FUNCTION_BLOCK Q_GraphicsContext (* Command Graphics Context ( Part 6 - F.56 ) *)
  (* Standard: ISO 11783-6; Description: Copyright (c) 2022 HR Agrartechnik GmbH This program and the accompanying materials are made available under the terms of the Eclipse Public License 2.0 which is available at https://www.eclipse.org/legal/epl-2.0/ SPDX-License-Identifier: EPL-2.0 see Description Tab *)
  (* Version 1.0, 2022-07-08, Franz Höpfinger, HR Agrartechnik GmbH *)
  PACKAGE isobus::UT::Q;
  IMPORT isobus::UT::Q::const::IDs::ID_NULL;
  (* Documentation:
  Command Graphics Context ( Part 6 - F.56 )
   This command is used to manipulate a graphics Context object (only on version 4 or later VTs).
   Valid Object IDs
   A graphics context Object ID is valid if it falls within the following ISO 11783-6 ID range:
    - GraphicsContextObject: 36000 – 36999
    ID_NULL (65535) is not a command target but can be used in INIT to deactivate the FB. Any ID outside this range is invalid for commanding.
   Activate / Deactivate
   The FB is deactivated by default. It becomes active when INIT provides a valid graphics context Object ID. Sending INIT with ID_NULL (65535) deactivates the FB again. This toggle can be repeated arbitrarily.
    - INIT + ID_NULL (65535): FB deactivated, STATUS="DEACTIVATED", s16result=VT_E_DEACTIVATED (-40)
   - INIT + valid graphics context ID: FB activated, STATUS="initialized", s16result=VT_E_NO_ERR (0). If a REQ was buffered before, it is executed immediately.
   - INIT + invalid ID: STATUS="ERROR: Invalid Object ID (not a graphics context object)", s16result=VT_E_INVALID_OBJECT_ID (-132)
    REQ Handling
    - REQ before any INIT: Buffered, STATUS="Buffered: INIT not yet completed", s16result=VT_E_NOT_READY (-131)
   - REQ while deactivated (INIT came with NULL or invalid ID): STATUS shows the actual deactivation reason, s16result=VT_E_DEACTIVATED (-40) or VT_E_INVALID_OBJECT_ID (-132)
   - REQ while active: Command sent to VT, result reflected in CNF
    param[in] {objectID, uint16_t}
   Object ID of a Graphics Context object. Use ID_NULL (65535) to deactivate the FB. Use a valid graphics context object ID to activate.
   param[in] {SubCommandID, uint8_t}
   Sub-Command ID
   param[in] {ParameterSubCommandID_Byte, const uint8_t *}
   Parameters based on sub-command ID byte
   param[in] {LenBytes, uint16_t}
   Length in bytes of parameter list
   Return Values (s16result):
   int16_t
    - VT_E_NO_ERR (0) - OK
   - VT_E_DEACTIVATED (-40) - FB deactivated (INIT received with ID_NULL)
   - VT_E_INVALID_OBJECT_ID (-132) - Object ID is invalid (not a graphics context object)
   - VT_E_NOT_READY (-131) - Buffered: INIT not yet completed
   - VT_E_OVERFLOW (-6) - buffer overflow
   - VT_E_NOACT (-8) - Command not possible in current state
   - VT_E_NO_INSTANCE (-21) - No VT client available
   - VT_E_ISO_INSTANCE_INVALID (-129) - Identifier for instance (connection) invalid
   - VT_E_NOT_ALIVE (-130) - Identifier for instance valid, but VT Dead.
    Note
    - Function uses string buffer ( Parameterlist has to be smaller than ISO_VTC_CMD_STR_MAX_LENGTH )
  *)
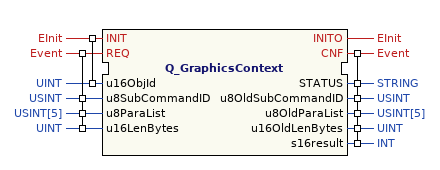
  EVENT_INPUT
    INIT : EInit WITH u16ObjId; (* Service Initialization *)
    REQ WITH u8SubCommandID, u8ParaList, u16LenBytes; (* Service Request *)
  END_EVENT
  EVENT_OUTPUT
    INITO : EInit; (* Initialization Confirm *)
    CNF WITH STATUS, s16result, u8OldSubCommandID, u8OldParaList, u16OldLenBytes; (* Confirmation of Requested Service *)
  END_EVENT
  VAR_INPUT
    u16ObjId : UINT := ID_NULL; (* Object ID *)
    u8SubCommandID : USINT; (* Sub-Command ID *)
    u8ParaList : ARRAY [0..4] OF USINT; (* Parameters based on sub-command ID byte *)
    u16LenBytes : UINT; (* Length in bytes of parameter list *)
  END_VAR
  VAR_OUTPUT
    STATUS : STRING; (* Service Status *)
    u8OldSubCommandID : USINT; (* Old Sub-Command ID *)
    u8OldParaList : ARRAY [0..4] OF USINT; (* Old parameters based on sub-command ID byte *)
    u16OldLenBytes : UINT; (* Old length in bytes of parameter list *)
    s16result : INT; (* retval see description *)
  END_VAR
END_FUNCTION_BLOCK
